// TIA Portal V18 export
TYPE "LGasp_type_Bck_visualizzazioni"
// stored: IsFailsafeCompliant false
   STRUCT
      visbool00 { ExternalWritable := 'False'} : Array[1..32] of Bool;
      visbool01 { ExternalAccessible := 'False'; ExternalVisible := 'False'; ExternalWritable := 'False'} : Array[1..32] of Bool;
      visbool02 { ExternalAccessible := 'False'; ExternalVisible := 'False'; ExternalWritable := 'False'} : Array[1..32] of Bool;
      visbool03 { ExternalAccessible := 'False'; ExternalVisible := 'False'; ExternalWritable := 'False'} : Array[1..32] of Bool;
      vis00 : DWord;
      vis01 : DWord;
      vis02 : DWord;
      vis03 : DWord;
      visint : Array[1..32] of Int;
      visdint : Array[1..32] of DInt;
      vislreal : Array[1..32] of LReal;
      visstring : Array[1..32] of WString;
   END_STRUCT;
   // // visbool00[1] : Trasferimento lista produzione in corso
   // // visbool00[2] : trasferimento valori DS
   // // visbool00[4] : Risposta pulsante PC svuotamento premuto
   // // visbool00[5] : Richiesta invio nuove righe di produzione
   // // visbool00[6] : 1 = Blocco modifiche righe di produzione/linea in marcia
   // // visbool00[7] : Risposta lista compilata
   // // visbool00[8] : abilitazione operazioni compilazione
   // // visbool00[9] : Abilita pulsante cancelli pezzi fatti
   // // visbool00[10] : Blocco totale modifica righe produzione
   // // visbool00[11] : Blocco input valore override profila
   // // visbool00[15] : Richiesta visualizzazione finestra inserimento lamiera
   // // visbool00[17] : Richiesta salvataggio correttori profila
   // // visbool00[19] : Approntamento profila eseguito
   // // visbool00[20] : Abilitazione comando sincronizzazione profila
   // // visbool00[21] : Abilitazione pulsante comando svuotamento scarico
   // // visbool00[22] : Risposta svuotamento scarico in corso
   // // visbool00[23] : Visualizzazione quota rimanente dell'ultimo pezzo da fare dopo l'allarme di fine lamiera (210100006/7 insieme a real 4)
   // // visbool00[30] : Svuotamento in corso
   // // visbool00[32] : Abilitazione pulsante svuotamento su PC
   // // visbool01[10] : Richiesta posizionamento stampo mobile P04 (210100012)
   // // visdint[1] : Totalizzatore assoluto pezzi fatti
   // // vislreal[1] : Velocità linea (m/min)
   // // vislreal[2] : Produttività linea (pz/min)
   // // vislreal[3] : Quota dopo lama (mm) 210100008
   // // vislreal[4] : Quota rimanente dell'ultimo pezzo da fare dopo l'allarme di fine lamiera (210100006/7 insieme a bool 23)
   // // vislreal[5] : Conteggio lunghezza materiale lavorato (km)
   // // vislreal[6] : Conteggio Ore linea accesa
   // // vislreal[7] : Conteggio Ore linea in automatico
   // // visstring[1] : Nome prodotto in lavoro
   // // visstring[2] : Nome prodotto in caricamento (durante approntamento linea)
END_TYPE
